FUNCTION_BLOCK EA_2_rightSwitch
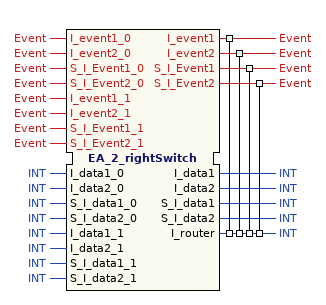
  EVENT_INPUT
    I_event1_0;
    I_event2_0;
    S_I_Event1_0;
    S_I_Event2_0;
    I_event1_1;
    I_event2_1;
    S_I_Event1_1;
    S_I_Event2_1;
  END_EVENT
  EVENT_OUTPUT
    I_event1 WITH I_router;
    I_event2 WITH I_router;
    S_I_Event1 WITH I_router;
    S_I_Event2 WITH I_router;
  END_EVENT
  VAR_INPUT
    I_data1_0 : INT;
    I_data2_0 : INT;
    S_I_data1_0 : INT;
    S_I_data2_0 : INT;
    I_data1_1 : INT;
    I_data2_1 : INT;
    S_I_data1_1 : INT;
    S_I_data2_1 : INT;
  END_VAR
  VAR_OUTPUT
    I_data1 : INT;
    I_data2 : INT;
    S_I_data1 : INT;
    S_I_data2 : INT;
    I_router : INT;
  END_VAR
  EC_STATES
    Start;
    I_event1_0_state : I_event1_0_algorithm -> I_event1;
    I_event2_0_state : I_event2_0_algorithm -> I_event2;
    S_I_Event1_0_state : S_I_Event1_0_algorithm -> S_I_Event1;
    S_I_Event2_0_state : S_I_Event2_0_algorithm -> S_I_Event2;
    I_event1_1_state : I_event1_1_algorithm -> I_event1;
    I_event2_1_state : I_event2_1_algorithm -> I_event2;
    S_I_Event1_1_state : S_I_Event1_1_algorithm -> S_I_Event1;
    S_I_Event2_1_state : S_I_Event2_1_algorithm -> S_I_Event2;
  END_STATES
  EC_TRANSITIONS
    I_event1_0_state TO Start := 1;
    Start TO I_event1_0_state := I_event1_0;
    I_event2_0_state TO Start := 1;
    Start TO I_event2_0_state := I_event2_0;
    S_I_Event1_0_state TO Start := 1;
    Start TO S_I_Event1_0_state := S_I_Event1_0;
    S_I_Event2_0_state TO Start := 1;
    Start TO S_I_Event2_0_state := S_I_Event2_0;
    I_event1_1_state TO Start := 1;
    Start TO I_event1_1_state := I_event1_1;
    I_event2_1_state TO Start := 1;
    Start TO I_event2_1_state := I_event2_1;
    S_I_Event1_1_state TO Start := 1;
    Start TO S_I_Event1_1_state := S_I_Event1_1;
    S_I_Event2_1_state TO Start := 1;
    Start TO S_I_Event2_1_state := S_I_Event2_1;
  END_TRANSITIONS
  ALGORITHM I_event1_0_algorithm IN ST:
I_data1 := I_data1_0;
I_data2 := I_data2_0;
S_I_data1 := S_I_data1_0;
S_I_data2 := S_I_data2_0;
I_router := 0;
  END_ALGORITHM
  ALGORITHM I_event2_0_algorithm IN ST:
I_data1 := I_data1_0;
I_data2 := I_data2_0;
S_I_data1 := S_I_data1_0;
S_I_data2 := S_I_data2_0;
I_router := 0;
  END_ALGORITHM
  ALGORITHM S_I_Event1_0_algorithm IN ST:
I_data1 := I_data1_0;
I_data2 := I_data2_0;
S_I_data1 := S_I_data1_0;
S_I_data2 := S_I_data2_0;
I_router := 0;
  END_ALGORITHM
  ALGORITHM S_I_Event2_0_algorithm IN ST:
I_data1 := I_data1_0;
I_data2 := I_data2_0;
S_I_data1 := S_I_data1_0;
S_I_data2 := S_I_data2_0;
I_router := 0;
  END_ALGORITHM
  ALGORITHM I_event1_1_algorithm IN ST:
I_data1 := I_data1_1;
I_data2 := I_data2_1;
S_I_data1 := S_I_data1_1;
S_I_data2 := S_I_data2_1;
I_router := 1;
  END_ALGORITHM
  ALGORITHM I_event2_1_algorithm IN ST:
I_data1 := I_data1_1;
I_data2 := I_data2_1;
S_I_data1 := S_I_data1_1;
S_I_data2 := S_I_data2_1;
I_router := 1;
  END_ALGORITHM
  ALGORITHM S_I_Event1_1_algorithm IN ST:
I_data1 := I_data1_1;
I_data2 := I_data2_1;
S_I_data1 := S_I_data1_1;
S_I_data2 := S_I_data2_1;
I_router := 1;
  END_ALGORITHM
  ALGORITHM S_I_Event2_1_algorithm IN ST:
I_data1 := I_data1_1;
I_data2 := I_data2_1;
S_I_data1 := S_I_data1_1;
S_I_data2 := S_I_data2_1;
I_router := 1;
  END_ALGORITHM
END_FUNCTION_BLOCK
